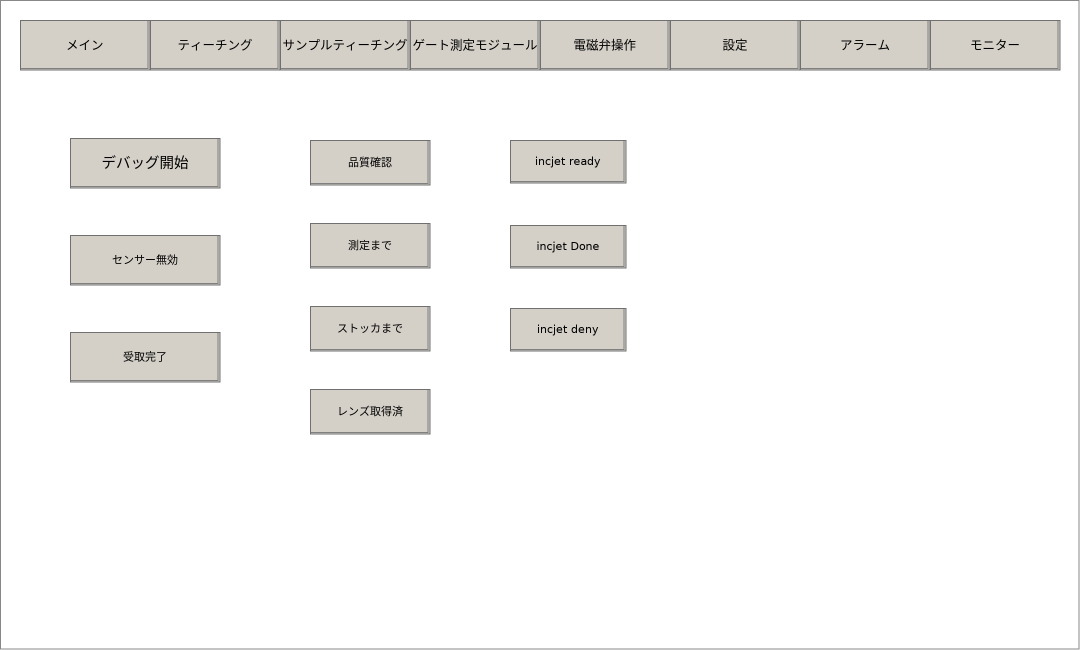
VISUALIZATION s_debug  // 1080x650
    Rectangle (0,0 1080x650)
    Button (20,20 130x50), "メイン"
        OnMouseClick: change screen: s_auto
    Button (150,20 130x50), "ティーチング"
        OnMouseClick: change screen: s_teaching1
    Button (670,20 130x50), "設定"
        OnMouseClick: change screen: s_setting
    Button (540,20 130x50), "電磁弁操作"
        OnMouseClick: change screen: s_manual
    Button (410,20 130x50), "ゲート測定モジュール"
        OnMouseClick: change screen: s_gm_teaching
    Button (800,20 130x50), "アラーム", colour toggle: gvl_io.flg_signalTowerRed
        OnMouseClick: change screen: s_alarm
    Button (280,20 130x50), "サンプルティーチング"
        OnMouseClick: change screen: s_sample
    Button (930,20 130x50), "モニター"
        OnMouseClick: change screen: s_monitor
    Button (70,235 150x50), "センサー無効", colour toggle: gvl_visu.flg_btn_vacSensOn, invisible if: NOT (gvl_debug.flg_debug_run AND gvl_param.var_currentMode = eP_programMode.auto), input disabled if: gvl_visu.flg_btn_vacSensOn
        toggle gvl_visu.flg_btn_vacSensOn
    Button (70,138 150x50), "デバッグ開始", colour toggle: gvl_debug.flg_debug_run, invisible if: NOT (gvl_param.var_currentMode = eP_programMode.auto), input disabled if: gvl_debug.flg_debug_run
        toggle gvl_debug.flg_debug_run
    Button (510,140 116x43), "incjet ready", colour toggle: gvl_debug.flg_stampReady, invisible if: NOT gvl_visu.flg_usingTimeStamp
        toggle gvl_debug.flg_stampReady
    Button (510,225 116x43), "incjet Done", colour toggle: gvl_debug.flg_stampDone, invisible if: NOT gvl_visu.flg_usingTimeStamp
        tap gvl_debug.flg_stampDone
    Button (510,308 116x43), "incjet deny", colour toggle: gvl_gm.var_incjetInfo.flg_denyStamp, invisible if: NOT gvl_visu.flg_usingTimeStamp
        toggle gvl_gm.var_incjetInfo.flg_denyStamp
    Button (310,223 120x45), "測定まで", colour toggle: gvl_debug.flg_to_measurement, invisible if: NOT (gvl_param.var_currentMode = eP_programMode.auto AND gvl_debug.flg_check_quality)
        toggle gvl_debug.flg_to_measurement
    Button (310,306 120x45), "ストッカまで", colour toggle: gvl_debug.flg_to_stocker, invisible if: NOT (gvl_param.var_currentMode = eP_programMode.auto AND gvl_debug.flg_check_quality)
        toggle gvl_debug.flg_to_stocker
    Button (310,389 120x45), "レンズ取得済", colour toggle: gvl_debug.flg_to_acquired, invisible if: NOT gvl_debug.flg_to_demand
        tap gvl_debug.flg_to_acquired
    Button (310,140 120x45), "品質確認", colour toggle: gvl_debug.flg_check_quality, invisible if: NOT (gvl_param.var_currentMode = eP_programMode.auto)
        toggle gvl_debug.flg_check_quality
    Button (70,332 150x50), "受取完了", invisible if: gvl_visu.flg_btn_vacSensOn OR NOT gvl_debug.out_busy OR NOT gvl_io.in_wire_gm_fiberSens
        tap gvl_visu.flg_btn_lensSetDone
END_VISUALIZATION

(* stored: Version 1.1.0.1, ProductVersion 3.1.4024.11
   Visu s_debug: Id {2b5719fb-3381-4cc2-825c-9b55c0761363} *)
